FUNCTION_BLOCK XtsHardwareTesting EXTENDS XtsHardware
VAR
	bExecute:		BOOL;
	fbTestsuites:	FB_Testsuites;				// Testsuites
	XtsHardwareTestSuite : FB_Testsuite;
	
	// Test-vars	

END_VAR

//// Run
//fbTestsuites();

//IF bExecute THEN
//	// manual execute | override file path
//	fbTestsuites.P_FilePathName:= 'C:\XtsHardwareTestReport.xml';
//	bExecute:= NOT fbTestsuites.M_Request(E_Base.Execute);
//END_IF

//// Add Testsuite to Testsuites
//fbTestsuites.M_Add(XtsHardwareTestSuite);

//{region "XtsRunnerTestSuite"}
//XtsHardwareTestSuite();
//CASE XtsHardwareTestSuite.P_Testcase OF
//	E_Testcase.Start:
//		FOR i := 1 TO SystemParameters.nModuleNumber DO
//			f24V[i] := 0;	 
//		END_FOR
//		XtsHardwareTestSuite.P_Assert.M_Equals_DINT(1,THIS^.Is24VOK(),'check the 24vdc reports low correctly');
//		XtsHardwareTestSuite.M_Testcase('XtsHardware',T#1S,'','',1);
//	1:
//		FOR i := 1 TO SystemParameters.nModuleNumber DO
//			f24V[i] := 24000;	 
//		END_FOR 
//		f24V[2] := 18000;
//		XtsHardwareTestSuite.P_Assert.M_Equals_DINT(1,THIS^.Is24VOK(),'check the 24vdc reports low correctly with single sensor');
//		XtsHardwareTestSuite.M_Testcase('XtsHardware',T#1S,'','',2);
//	2:
//		FOR i := 1 TO SystemParameters.nModuleNumber DO
//			f24V[i] := 24000;	 
//		END_FOR  
//		XtsHardwareTestSuite.P_Assert.M_Equals_DINT(2,THIS^.Is24VOK(),'check the 24vdc reports 24vdcok correctly');
//		XtsHardwareTestSuite.M_Testcase('XtsHardware',T#1S,'','',3);
//	3:
//		 FOR i := 1 TO SystemParameters.nModuleNumber DO
//			f24V[i] := 29000;	 
//		END_FOR  
//		XtsHardwareTestSuite.P_Assert.M_Equals_DINT(1,THIS^.Is24VOK(),'check the 24vdc reports 24vdcok correctly');
//		XtsHardwareTestSuite.M_Testcase('XtsHardware',T#1S,'','',4);
//	4:
//		 FOR i := 1 TO SystemParameters.nModuleNumber DO
//			f24V[i] := 24000;	 
//		END_FOR  
//		f24V[2] := 29000;
//		XtsHardwareTestSuite.P_Assert.M_Equals_DINT(1,THIS^.Is24VOK(),'check the 24vdc reports 24vdcok correctly');
//		XtsHardwareTestSuite.M_Testcase('XtsHardware',T#1S,'','',5);
	
//	5:
//		FOR i := 1 TO SystemParameters.nModuleNumber DO
//			f48V[i] := 0;	 
//		END_FOR
//		XtsHardwareTestSuite.P_Assert.M_Equals_DINT(1,THIS^.Is48VOK(),'check the 24vdc reports low correctly');
//		XtsHardwareTestSuite.M_Testcase('XtsHardware',T#1S,'','',6);
//	6:
//		FOR i := 1 TO SystemParameters.nModuleNumber DO
//			f48V[i] := 48000;	 
//		END_FOR 
//		f48V[2] := 46000;
//		XtsHardwareTestSuite.P_Assert.M_Equals_DINT(1,THIS^.Is48VOK(),'check the 24vdc reports low correctly with single sensor');
//		XtsHardwareTestSuite.M_Testcase('XtsHardware',T#1S,'','',7);
//	7:
//		FOR i := 1 TO SystemParameters.nModuleNumber DO
//			f48V[i] := 48000;	 
//		END_FOR  
//		XtsHardwareTestSuite.P_Assert.M_Equals_DINT(2,THIS^.Is48VOK(),'check the 24vdc reports 24vdcok correctly');
//		XtsHardwareTestSuite.M_Testcase('XtsHardware',T#1S,'','',8);
//	8:
//		 FOR i := 1 TO SystemParameters.nModuleNumber DO
//			f48V[i] := 50000;	 
//		END_FOR  
//		XtsHardwareTestSuite.P_Assert.M_Equals_DINT(1,THIS^.Is48VOK(),'check the 24vdc reports 24vdcok correctly');
//		XtsHardwareTestSuite.M_Testcase('XtsHardware',T#1S,'','',9);
//	9:
//		 FOR i := 1 TO SystemParameters.nModuleNumber DO
//			f48V[i] := 48000;	 
//		END_FOR  
//		f48V[2] := 50000;
//		XtsHardwareTestSuite.P_Assert.M_Equals_DINT(1,THIS^.Is48VOK(),'check the 24vdc reports 24vdcok correctly');
//		XtsHardwareTestSuite.M_Testcase('XtsHardware',T#1S,'','',E_Testcase.Done);

//	E_Testcase.Done:;
		 
//END_CASE
//{endregion}

END_FUNCTION_BLOCK

(* stored: Version 1.1.0.1, ProductVersion 3.1.4024.12
   POU XtsHardwareTesting: Id {7afd002c-75a0-46c4-9267-fe0bdcc43af0}, SpecialFunc None *)
